ABB RAPID module: 0028F5F2

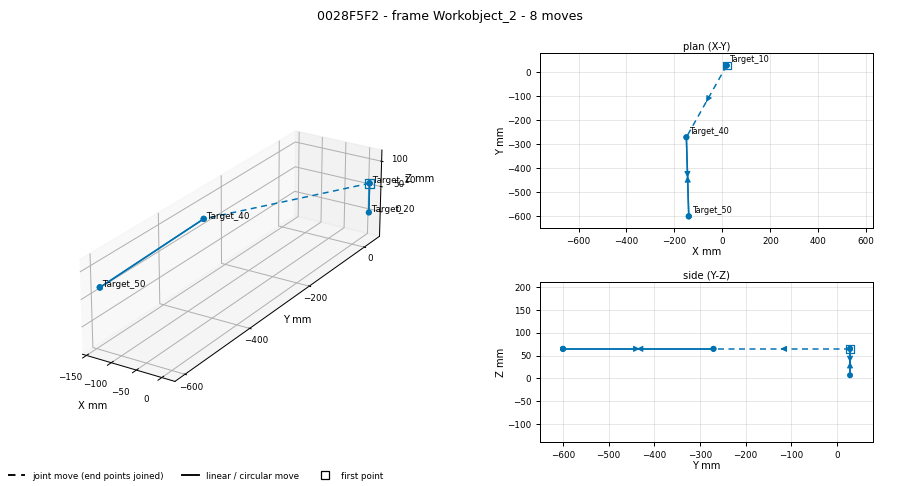
[picture p0: tool path of 0028F5F2 in frame Workobject_2, 8 of 8 moves have a stored position in this frame; points joined in program order, loops and branches not executed]
MODULE Module1
        CONST robtarget Target_10:=[[17.680006378,29.000003785,64.999943406],[-0.000000006,1,0,0.000000004],[-1,0,-1,0],[9E+09,9E+09,9E+09,9E+09,9E+09,9E+09]];
    CONST robtarget Target_20:=[[17.680005,29.000006044,6.999955902],[0.000000007,1,0,-0.000000004],[-1,-1,-1,0],[9E+09,9E+09,9E+09,9E+09,9E+09,9E+09]];
    CONST robtarget Target_30:=[[17.680006378,29.000003785,64.999943406],[-0.000000006,1,0,0.000000004],[-1,0,-1,0],[9E+09,9E+09,9E+09,9E+09,9E+09,9E+09]];
    CONST robtarget Target_40:=[[-150.200005115,-270.140000008,64.999941394],[-0.000000007,0.871855665,0.489762902,0.000000004],[0,0,-1,0],[9E+09,9E+09,9E+09,9E+09,9E+09,9E+09]];
    CONST robtarget Target_50:=[[-140.200013899,-600.000004341,64.999949592],[0.000000013,0.871855673,0.489762887,0.000000004],[0,-1,-1,0],[9E+09,9E+09,9E+09,9E+09,9E+09,9E+09]];
    CONST robtarget Target_60:=[[-140.200013899,-600.000004341,64.999949592],[0.000000014,0.707106787,0.707106776,0],[0,-1,-1,0],[9E+09,9E+09,9E+09,9E+09,9E+09,9E+09]];
    VAR num contador :=0;
!***********************************************************
    !
    ! Módulo:  Module1
    !
    ! Descripción:
    !   <Introduzca la descripción aquí>
    !
    ! Autor: Admin
    !
    ! Versión: 1.0
    !
    !***********************************************************


    !***********************************************************
    !
    ! Procedimiento Main
    !
    !   Este es el punto de entrada de su programa
    !
    !***********************************************************
    PROC main()
        !Añada aquí su código
        setDO Start6_Controlador, 0;
        setDO Start10_Controlador, 0;
        setDO Start12_Controlador, 0;
        ciclo_inicio_tenedor:
        IF cajas_6=high THEN
            setDO Start6_Controlador, 1;
            !setDO Start6_Controlador, 0;
            contador :=6;
            Rutina_tenedor;
        ELSEIF cajas_10=high THEN
            setDO Start10_Controlador, 1;
            !setDO Start10_Controlador, 0;
            contador :=10;
            Rutina_tenedor;
        ELSEIF cajas_12=high THEN
            setDO Start12_Controlador, 1;
            !setDO Start12_Controlador, 0;
            contador :=12;
            Rutina_tenedor;
        ELSE
            GOTO ciclo_inicio_tenedor;
        ENDIF

    ENDPROC
    PROC Rutina_tenedor()
        WHILE contador>0 DO
            WaitDI CajaOK,1;
            WaitDI CucharaOK,1;
            WaitDI TenedorOK,1;
            MoveJ Target_10,v600,z10,TCP_Ventosa\WObj:=Workobject_2;
            MoveL Target_20,v150,z1,TCP_Ventosa\WObj:=Workobject_2;
            MoveL Target_30,v150,z1,TCP_Ventosa\WObj:=Workobject_2;
            MoveJ Target_40,v600,z10,TCP_Ventosa\WObj:=Workobject_2;
            MoveL Target_50,v300,z1,TCP_Ventosa\WObj:=Workobject_2;
            MoveL Target_60,v300,z1,TCP_Ventosa\WObj:=Workobject_2;
            MoveL Target_50,v300,z1,TCP_Ventosa\WObj:=Workobject_2;
            MoveL Target_40,v300,z1,TCP_Ventosa\WObj:=Workobject_2;
            contador := contador-1;
        ENDWHILE
    ENDPROC
ENDMODULE
